FUNCTION_BLOCK FB_ShutDown
VAR_INPUT
	fbUPS			:iUPS;				// UPS interface	
END_VAR
VAR_OUTPUT
END_VAR
VAR
	eShutdownMode	:E_ShutdownMode;	// State machine when shutting down
END_VAR

// watch power fail
fbUPS.watch_status();

CASE fbUPS.UPSState OF 
	E_UPSState.on_battery:
		eShutdownMode := E_ShutdownMode.persistent_data;
	E_UPSState.critical_error:
		eShutdownMode := E_ShutdownMode.shutting_down;
	ELSE
		eShutdownMode := E_ShutdownMode.init;
END_CASE

CASE eShutdownMode OF 
	E_ShutdownMode.persistent_data:
		fbUPS.persist_data();
		IF fbUPS.UPSState = E_UPSState.facility_error THEN
			eShutdownMode := E_ShutdownMode.shutting_down;
		END_IF
	E_ShutdownMode.shutting_down:
		fbUPS.shutdown();
END_CASE

END_FUNCTION_BLOCK

(* stored: Version 1.1.0.1, ProductVersion 3.1.4024.12
   POU FB_ShutDown: Id {107fb3ae-5c98-443d-9a22-030f2796c1b3}, SpecialFunc None *)
